{attribute 'linkalways'} 
{attribute 'no_explicit_call' := 'This FB is a CLASS and must be accessed using methods or properties'}
{attribute 'enable_dynamic_creation'}
FUNCTION_BLOCK _ETcVnSvm EXTENDS EnumDatatypeBase
VAR
	localData : ETcVnSvm;
	activeData : REFERENCE TO ETcVnSvm;
	enumBaseDatatype : _UDINT(localData);
END_VAR

METHOD PRIVATE AddLocalEnumeration
VAR_INPUT
	Enumeration : T_MAXSTRING;
	Value : ETcVnSvm;
END_VAR
AddEnumeration(Enumeration, Value);
END_METHOD

PROPERTY PUBLIC Address : PVOID
GET
Address := ADR(activeData);
END_GET
END_PROPERTY

METHOD PUBLIC ClearReference
VAR_INPUT
END_VAR
activeData REF= localData;
SetBaseDatatypeReference();
END_METHOD

METHOD PUBLIC Clone : I_Datatype
VAR
    pClone : POINTER TO _ETcVnSvm;
END_VAR
pClone := __NEW(_ETcVnSvm(InitialValue := Value));
Clone := pClone^;
END_METHOD

METHOD FB_init : BOOL
VAR_INPUT
	bInitRetains : BOOL; // if TRUE, the retain variables are initialized (warm start / cold start)
	bInCopyCode : BOOL;  // if TRUE, the instance afterwards gets moved into the copy code (online change)
	InitialValue : ETcVnSvm;
END_VAR
localData := InitialValue;
AddBaseDatatype(enumBaseDatatype);
ClearReference();

AddLocalEnumeration('TCVN_SVM_C_CLASSIFIER', ETcVnSvm.TCVN_SVM_C_CLASSIFIER);
AddLocalEnumeration('TCVN_SVM_NU_CLASSIFIER', ETcVnSvm.TCVN_SVM_NU_CLASSIFIER);
AddLocalEnumeration('TCVN_SVM_NOVELTY_DETECTOR', ETcVnSvm.TCVN_SVM_NOVELTY_DETECTOR);
AddLocalEnumeration('TCVN_SVM_EPS_REGRESSOR', ETcVnSvm.TCVN_SVM_EPS_REGRESSOR);
AddLocalEnumeration('TCVN_SVM_NU_REGRESSOR', ETcVnSvm.TCVN_SVM_NU_REGRESSOR);
END_METHOD

PROPERTY PUBLIC Identifier : T_MAXSTRING
GET
Identifier := 'ETcVnSvm';
END_GET
END_PROPERTY

METHOD IsEnumeratorValueEqual : BOOL
VAR_INPUT
	Enumerator : I_KeyValueForwardEnumerator;
END_VAR
VAR
	storedValue : ETcVnSvm;
END_VAR
IF NOT Enumerator.TryGet(storedValue) THEN
	RETURN;
END_IF

IsEnumeratorValueEqual := storedValue = activeData;
END_METHOD

METHOD PUBLIC MakeReferenceTo
VAR_INPUT
	ReferenceTarget : REFERENCE TO ETcVnSvm;
END_VAR
activeData REF= ReferenceTarget;
SetBaseDatatypeReference();
END_METHOD

METHOD PROTECTED SetBaseDatatypeReference
VAR_INPUT
END_VAR
enumBaseDatatype.MakeReferenceTo(activeData);
END_METHOD

PROPERTY PUBLIC Size : UDINT
GET
Size := SIZEOF(activeData);
END_GET
END_PROPERTY

METHOD TryMakeReferenceTo : BOOL
VAR_INPUT
	Target : I_Datatype;
END_VAR
VAR
	targetAsEnum : I_EnumDatatype;
	pTargetData : POINTER TO ETcVnSvm;
END_VAR
IF NOT Target.TryResolveAsEnumDatatype(targetAsEnum) THEN
	RETURN;
END_IF

IF targetAsEnum.Identifier <> Identifier THEN
	RETURN;
END_IF

pTargetData := Target.Address;
activeData REF= pTargetData^;
SetBaseDatatypeReference();
TryMakeReferenceTo := TRUE;
END_METHOD

PROPERTY PUBLIC Value : ETcVnSvm
GET
Value := activeData;
END_GET
SET
activeData := Value;
END_SET
END_PROPERTY

END_FUNCTION_BLOCK

(* stored: Version 1.1.0.1, ProductVersion 3.1.4024.12
   POU _ETcVnSvm: Id {001a7d7a-217d-07c7-25f0-bba8896458c6}, SpecialFunc None
   Folder Constructor: Id {6c4341a2-2408-0980-021d-8d97d8e0bee7}
   Folder Private: Id {f165579c-a59b-007e-02dd-61653742256b}
   Folder Protected: Id {932db8f1-2661-00f0-2a77-ffeec83a3186}
   Method AddLocalEnumeration: Id {8c6957d9-8ceb-0bcb-0fd4-f3f8dfecaa73}
   Property Address: Id {dd758ee0-9de3-0c7b-30a0-0bf288820bd5}
   Get Get: Id {38636242-11ab-03a6-199c-020e7b6cf7cd}
   Method ClearReference: Id {6e371719-af13-0923-3061-be284cafa58f}
   Method Clone: Id {90ce5e0f-79c2-093e-0c3f-e293b0a6dcde}
   Method FB_init: Id {cc1b0afe-bcdd-0c1b-0e97-706daa50fd82}
   Property Identifier: Id {38a59a1e-04f6-0e22-21fd-49256d135e56}
   Get Get: Id {35b2f522-10fc-0512-3271-e778d9b7b044}
   Method IsEnumeratorValueEqual: Id {3855992b-0315-0688-3bda-2a9e4d5c851c}
   Method MakeReferenceTo: Id {09f6ca40-126c-0d05-197b-55bfa124a765}
   Method SetBaseDatatypeReference: Id {41662b47-d241-0100-3701-b5fc4cf8309a}
   Property Size: Id {3ef816e2-a389-0e96-302a-62452d083275}
   Get Get: Id {08b533c7-1f58-0a2f-0754-1af32d4388af}
   Method TryMakeReferenceTo: Id {dbee9c29-ccb2-06bb-2427-894d407d21ea}
   Property Value: Id {dfa17475-5e7b-059c-32ee-2ae91d8f6096}
   Get Get: Id {584daca3-0f90-04c5-19eb-7a5e6d097013}
   Set Set: Id {e1972abd-a55f-00ed-1c93-3d2ce35d2740} *)
